FUNCTION_BLOCK FB_LoadWeight
VAR_INPUT
	stLoadIn			:ST_LoadData;
	bEnable				:BOOL;
	iConvStatus			:BYTE;
	bAutomat			:BOOL;
	
	rInWeight			:DINT;;
	bMove				:BOOL;
	bReadWeight     	:BOOL;
	
	bResetCTUWeight		:BOOL;	//Очистка счетчика невзвешиваний	
	bSetValWeight		:WORD;	//Заданное значение разрешенных ошибок
END_VAR
VAR_OUTPUT
	bEnableReadyData	:BOOL;
	bRequestWeight		:BOOL;
	bCountNoReadWeight	:WORD;		//Кол-во несчитываний
	bOverflowWeight		:BOOL;		//Переполнение счетчика несчитываний весов
END_VAR
VAR
	fbPulsRequest		:R_TRIG;
	bStartRequest		:BOOL;
	fbPulsReadWeight	:R_TRIG;
	fbDelayWeight		:TON;
	fbStartMove			:R_TRIG;
	fbFinMove			:F_TRIG;
	bReadySt			:BOOL;
	bStartMove			:BOOL;
	bEndMove			:BOOL;
	sInWeight			:STRING;
	
	WaitingWeight		:TON;
	bNoReadWeight		:BOOL;		//Несчитывание
	bWriteWeightGood	:BOOL;
	fbPulsNoreadWeight 	:R_TRIG;
	CTU 				:CTU;		//Счетчик
END_VAR

VAR_IN_OUT
	stLoadMove      	:ST_LoadData;
	stLoad				:ST_LoadData;
//	bReadWeight			:BOOL;
END_VAR

fbStartMove(CLK:=bMove);
bStartMove S=fbStartMove.Q;
IF bStartMove THEN 
	stLoadMove := stLoadIn;
	IF stLoadMove.sID=stLoadIn.sID  AND stLoadMove.sWeight=stLoadIn.sWeight  THEN
		bStartMove:=FALSE;
	END_IF
END_IF

fbFinMove(CLK:=bMove);
bEndMove S= fbFinMove.Q;
IF bEndMove THEN 
	stLoad := stLoadMove;
	IF stLoadMove.sID=stLoad.sID  AND stLoadMove.sWeight=stLoad.sWeight  THEN
		bEndMove:=FALSE;
	END_IF
END_IF
//bReadySt := stLoad.sID = stLoadIn.sID  AND stLoad.sWeight = stLoadIn.sWeight;

bStartRequest:= bEnable AND bAutomat AND (iConvStatus=2 OR iConvStatus=3) AND NOT bEndMove;

bEnableReadyData 	R= NOT bStartRequest;
bRequestWeight 		R= NOT bStartRequest;
bNoReadWeight		R= NOT bStartRequest;

fbPulsRequest(CLK:=bStartRequest);
IF fbPulsRequest.Q THEN
	bRequestWeight:=TRUE;
END_IF

WaitingWeight(IN:= bRequestWeight, PT:=T#2S);
bNoReadWeight S= WaitingWeight.Q ;

fbPulsNoreadWeight(CLK:=bNoReadWeight);

CTU(CU:=fbPulsNoreadWeight.Q, RESET:=bResetCTUWeight, PV:=bSetValWeight);
bCountNoReadWeight:=CTU.CV;

fbDelayWeight(IN:=bRequestWeight(*bReadWeight*), PT:=T#0.3S);

sInWeight:= DINT_TO_STRING(rInWeight);
IF bRequestWeight(*bReadWeight  AND bReadySt*)AND NOT (bCountNoReadWeight=bSetValWeight) THEN
	stLoad.sWeight:= sInWeight;
	
	IF stLoad.sWeight<>'' OR fbDelayWeight.Q THEN	
		bWriteWeightGood	:=TRUE;	
		bRequestWeight		:=FALSE;
	END_IF	
END_IF

bEnableReadyData S= bWriteWeightGood OR bNoReadWeight;

IF iConvStatus=0 THEN
	stLoad.sID:= '';
	stLoad.sWeight:= '';
END_IF

IF bCountNoReadWeight>=bSetValWeight THEN bOverflowWeight:=TRUE;
	ELSE bOverflowWeight:=FALSE;
END_IF

END_FUNCTION_BLOCK

(* stored: Version 1.1.0.1, ProductVersion 3.1.4024.4
   POU FB_LoadWeight: Id {85719c14-b34b-437b-99eb-10e6232a4f30}, SpecialFunc None *)
